Staubli VAL3: print.pgx

program print(string line)
begin
  strStatus = line
  delay(0.5)
end
